DATA_BLOCK "Data_block_1"
{ S7_Optimized_Access := 'TRUE' }
NAME : '1'
VERSION : 0.1
NON_RETAIN
   VAR
      TagName1 : Bool;
      TagName2 : Byte;
      Motor1 { S7_SetPoint := 'False'} : "UDT_MOTOR";
   END_VAR

BEGIN

END_DATA_BLOCK
